Fanuc KAREL source: pos_cnvcart.kl

PROGRAM pos_cnvcart
%NOBUSYLAMP
%NOLOCKGROUP

VAR
	reg_no : INTEGER
	grp_no : INTEGER
%from tpe.klh %import get_int_arg
%from pose.klh %import matrix_to_cart

BEGIN
	reg_no = tpe__get_int_arg(1)
	grp_no = tpe__get_int_arg(2)
	pose__matrix_to_cart(reg_no,grp_no)
END pos_cnvcart
